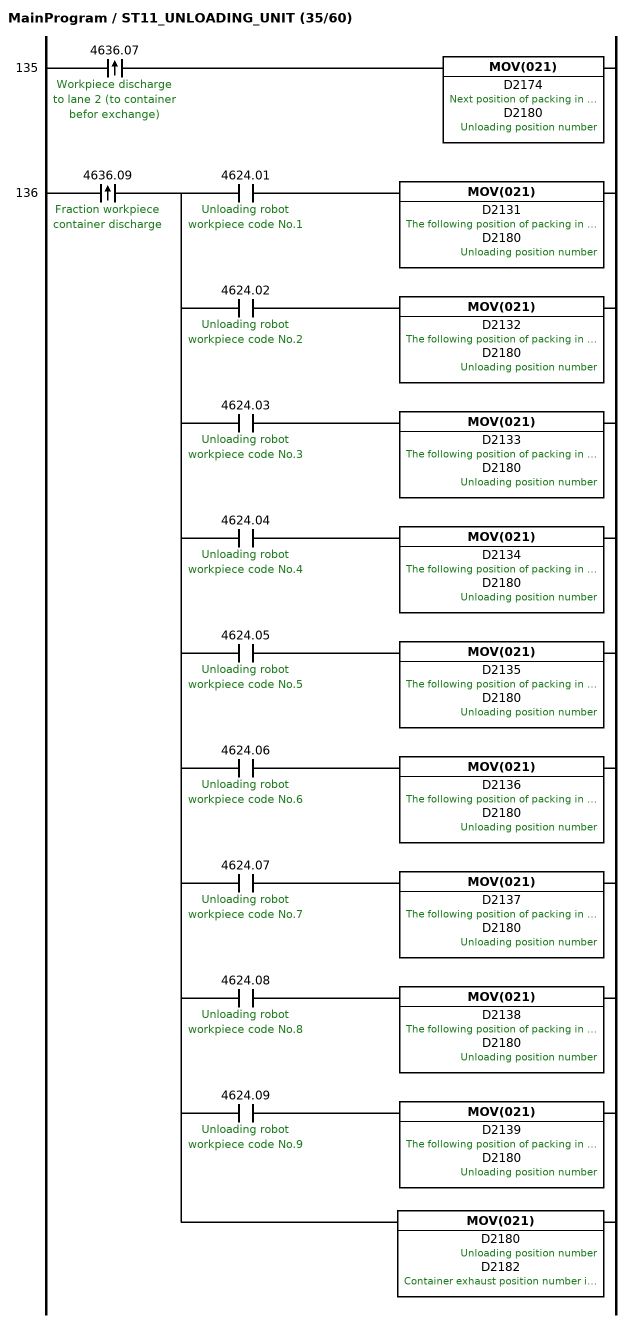
; [picture p552: MainProgram / ST11_UNLOADING_UNIT, rungs 135-136]
; rung 135
@LD 4636.07  ; Workpiece discharge to lane 2 (to container befor exchange)
MOV(021) D2174 D2180  ; Next position of packing in a container of lane 4 (exchange container)(BIN), Unloading position number
; rung 136
@LD 4636.09  ; Fraction workpiece container discharge
OUT TR0
AND 4624.01  ; Unloading robot workpiece code No.1
MOV(021) D2131 D2180  ; The following position of packing in a container number in fraction workpiece (code no.1), Unloading position number
LD TR0
AND 4624.02  ; Unloading robot workpiece code No.2
MOV(021) D2132 D2180  ; The following position of packing in a container number in fraction workpiece (code no.2), Unloading position number
LD TR0
AND 4624.03  ; Unloading robot workpiece code No.3
MOV(021) D2133 D2180  ; The following position of packing in a container number in fraction workpiece (code no.3), Unloading position number
LD TR0
AND 4624.04  ; Unloading robot workpiece code No.4
MOV(021) D2134 D2180  ; The following position of packing in a container number in fraction workpiece (code no.4), Unloading position number
LD TR0
AND 4624.05  ; Unloading robot workpiece code No.5
MOV(021) D2135 D2180  ; The following position of packing in a container number in fraction workpiece (code no.5), Unloading position number
LD TR0
AND 4624.06  ; Unloading robot workpiece code No.6
MOV(021) D2136 D2180  ; The following position of packing in a container number in fraction workpiece (code no.6), Unloading position number
LD TR0
AND 4624.07  ; Unloading robot workpiece code No.7
MOV(021) D2137 D2180  ; The following position of packing in a container number in fraction workpiece (code no.7), Unloading position number
LD TR0
AND 4624.08  ; Unloading robot workpiece code No.8
MOV(021) D2138 D2180  ; The following position of packing in a container number in fraction workpiece (code no.8), Unloading position number
LD TR0
AND 4624.09  ; Unloading robot workpiece code No.9
MOV(021) D2139 D2180  ; The following position of packing in a container number in fraction workpiece (code no.9), Unloading position number
LD TR0
MOV(021) D2180 D2182  ; Unloading position number, Container exhaust position number in fraction workpiece

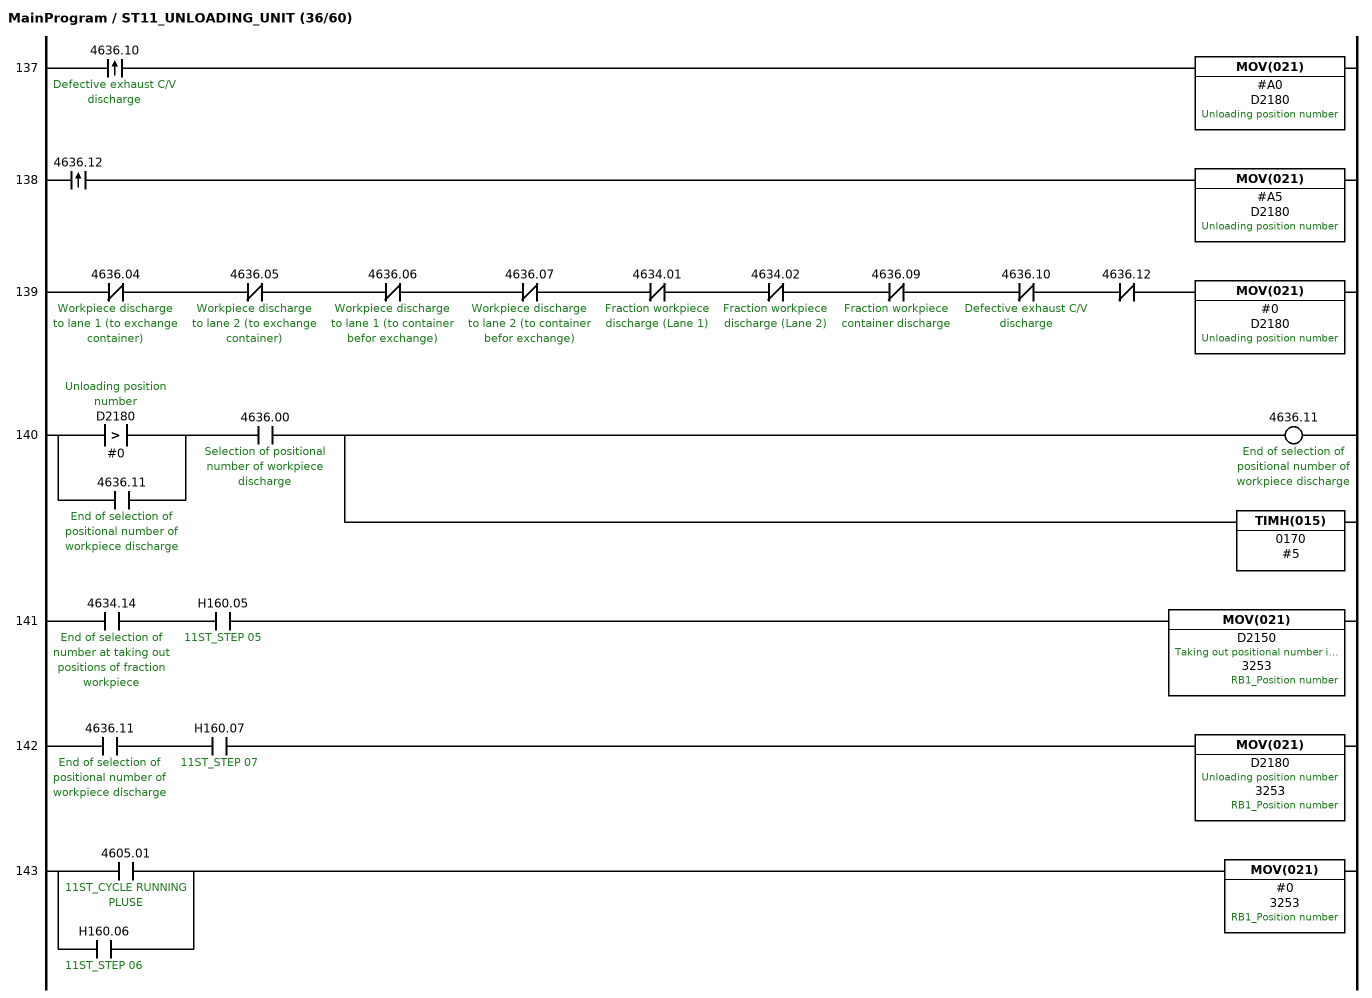
; rung 137
@LD 4636.10  ; Defective exhaust C/V discharge
MOV(021) #A0 D2180  ; Unloading position number
; rung 138
@LD 4636.12
MOV(021) #A5 D2180  ; Unloading position number
; rung 139
LDNOT 4636.04  ; Workpiece discharge to lane 1 (to exchange container)
ANDNOT 4636.05  ; Workpiece discharge to lane 2 (to exchange container)
ANDNOT 4636.06  ; Workpiece discharge to lane 1 (to container befor exchange)
ANDNOT 4636.07  ; Workpiece discharge to lane 2 (to container befor exchange)
ANDNOT 4634.01  ; Fraction workpiece discharge (Lane 1)
ANDNOT 4634.02  ; Fraction workpiece discharge (Lane 2)
ANDNOT 4636.09  ; Fraction workpiece container discharge
ANDNOT 4636.10  ; Defective exhaust C/V discharge
ANDNOT 4636.12
MOV(021) #0 D2180  ; Unloading position number
; rung 140
LD>(320) D2180 #0  ; Unloading position number
OR 4636.11  ; End of selection of positional number of workpiece discharge
AND 4636.00  ; Selection of positional number of workpiece discharge
OUT 4636.11  ; End of selection of positional number of workpiece discharge
TIMH(015) 0170 #5
; rung 141
LD 4634.14  ; End of selection of number at taking out positions of fraction workpiece
AND H160.05  ; 11ST_STEP 05
MOV(021) D2150 3253  ; Taking out positional number in fraction workpiece, RB1_Position number
; rung 142
LD 4636.11  ; End of selection of positional number of workpiece discharge
AND H160.07  ; 11ST_STEP 07
MOV(021) D2180 3253  ; Unloading position number, RB1_Position number
; rung 143
LD 4605.01  ; 11ST_CYCLE RUNNING PLUSE
OR H160.06  ; 11ST_STEP 06
MOV(021) #0 3253  ; RB1_Position number

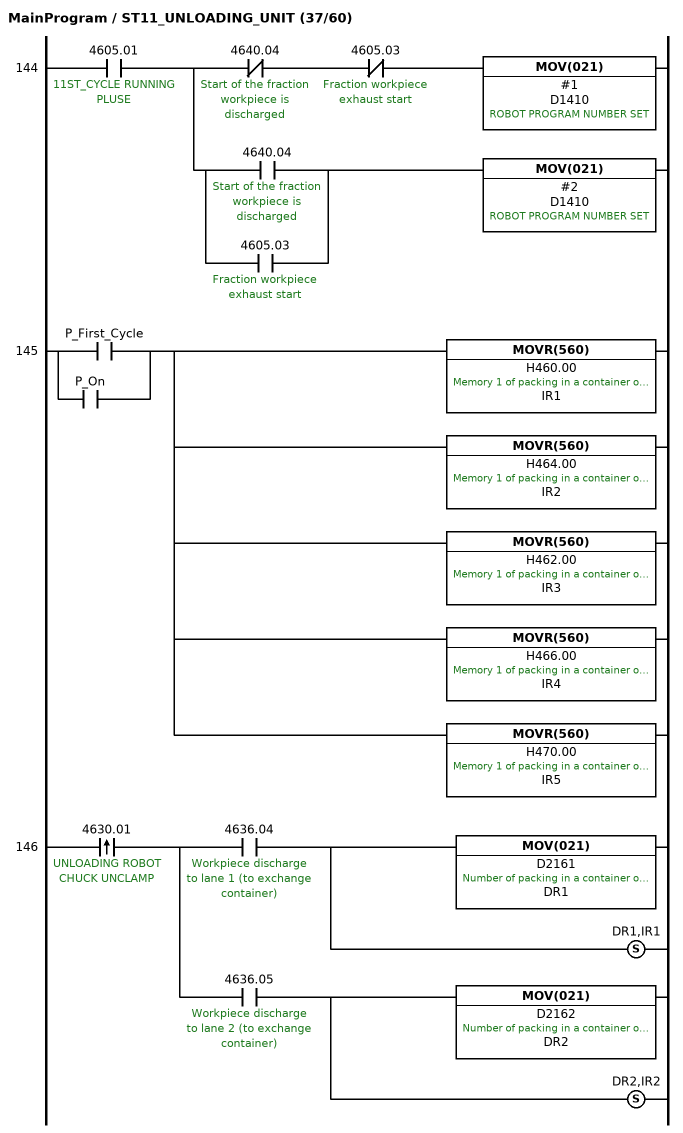
; rung 144
LD 4605.01  ; 11ST_CYCLE RUNNING PLUSE
OUT TR0
ANDNOT 4640.04  ; Start of the fraction workpiece is discharged
ANDNOT 4605.03  ; Fraction workpiece exhaust start
MOV(021) #1 D1410  ; ROBOT PROGRAM NUMBER SET
LD TR0
LD 4640.04  ; Start of the fraction workpiece is discharged
OR 4605.03  ; Fraction workpiece exhaust start
ANDLD
MOV(021) #2 D1410  ; ROBOT PROGRAM NUMBER SET
; rung 145
LD P_First_Cycle
OR P_On  // 様子見で入れた 070619
MOVR(560) H460.00 IR1  ; Memory 1 of packing in a container of lane 1 (exchange container)
MOVR(560) H464.00 IR2  ; Memory 1 of packing in a container of lane 2 (exchange container)
MOVR(560) H462.00 IR3  ; Memory 1 of packing in a container of lane 1 (container befor exchange)
MOVR(560) H466.00 IR4  ; Memory 1 of packing in a container of lane 2 (container befor exchange)
MOVR(560) H470.00 IR5  ; Memory 1 of packing in a container of fraction workpiece
; rung 146
@LD 4630.01  ; UNLOADING ROBOT CHUCK UNCLAMP
OUT TR0
AND 4636.04  ; Workpiece discharge to lane 1 (to exchange container)
MOV(021) D2161 DR1  ; Number of packing in a container of lane 1 (exchange container)(BIN)
SET DR1,IR1
LD TR0
AND 4636.05  ; Workpiece discharge to lane 2 (to exchange container)
MOV(021) D2162 DR2  ; Number of packing in a container of lane 2 (exchange container)(BIN)
SET DR2,IR2

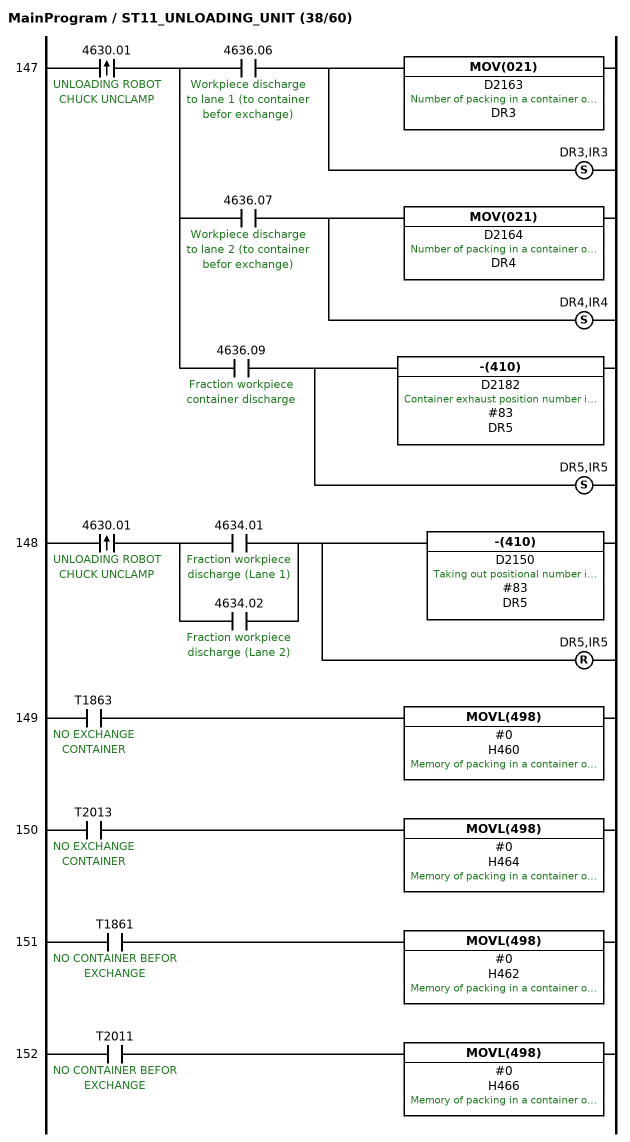
; rung 147
@LD 4630.01  ; UNLOADING ROBOT CHUCK UNCLAMP
OUT TR0
AND 4636.06  ; Workpiece discharge to lane 1 (to container befor exchange)
MOV(021) D2163 DR3  ; Number of packing in a container of lane 1 (container before exchange)(BIN)
SET DR3,IR3
LD TR0
AND 4636.07  ; Workpiece discharge to lane 2 (to container befor exchange)
MOV(021) D2164 DR4  ; Number of packing in a container of lane 2 (container before exchange)(BIN)
SET DR4,IR4
LD TR0
AND 4636.09  ; Fraction workpiece container discharge
-(410) D2182 #83 DR5  ; Container exhaust position number in fraction workpiece
SET DR5,IR5
; rung 148
@LD 4630.01  ; UNLOADING ROBOT CHUCK UNCLAMP
LD 4634.01  ; Fraction workpiece discharge (Lane 1)
OR 4634.02  ; Fraction workpiece discharge (Lane 2)
ANDLD
-(410) D2150 #83 DR5  ; Taking out positional number in fraction workpiece
RSET DR5,IR5
; rung 149
LD T1863  ; NO EXCHANGE CONTAINER
MOVL(498) #0 H460  ; Memory of packing in a container of lane 1 (exchange container)
; rung 150
LD T2013  ; NO EXCHANGE CONTAINER
MOVL(498) #0 H464  ; Memory of packing in a container of lane 2 (exchange container)
; rung 151
LD T1861  ; NO CONTAINER BEFOR EXCHANGE
MOVL(498) #0 H462  ; Memory of packing in a container of lane 1 (container befor exchange)
; rung 152
LD T2011  ; NO CONTAINER BEFOR EXCHANGE
MOVL(498) #0 H466  ; Memory of packing in a container of lane 2 (container befor exchange)

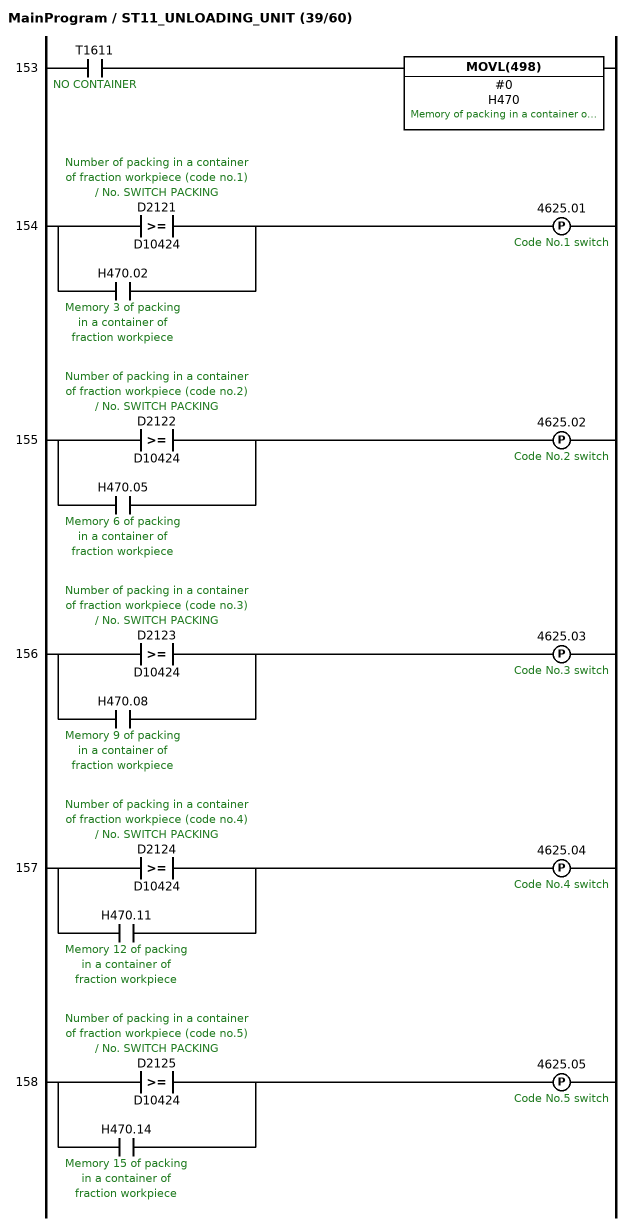
; rung 153
LD T1611  ; NO CONTAINER
MOVL(498) #0 H470  ; Memory of packing in a container of fraction workpiece
; rung 154
LD>=(325) D2121 D10424  ; Number of packing in a container of fraction workpiece (code no.1), No. SWITCH PACKING
OR H470.02  ; Memory 3 of packing in a container of fraction workpiece
DIFU(013) 4625.01  ; Code No.1 switch
; rung 155
LD>=(325) D2122 D10424  ; Number of packing in a container of fraction workpiece (code no.2), No. SWITCH PACKING
OR H470.05  ; Memory 6 of packing in a container of fraction workpiece
DIFU(013) 4625.02  ; Code No.2 switch
; rung 156
LD>=(325) D2123 D10424  ; Number of packing in a container of fraction workpiece (code no.3), No. SWITCH PACKING
OR H470.08  ; Memory 9 of packing in a container of fraction workpiece
DIFU(013) 4625.03  ; Code No.3 switch
; rung 157
LD>=(325) D2124 D10424  ; Number of packing in a container of fraction workpiece (code no.4), No. SWITCH PACKING
OR H470.11  ; Memory 12 of packing in a container of fraction workpiece
DIFU(013) 4625.04  ; Code No.4 switch
; rung 158
LD>=(325) D2125 D10424  ; Number of packing in a container of fraction workpiece (code no.5), No. SWITCH PACKING
OR H470.14  ; Memory 15 of packing in a container of fraction workpiece
DIFU(013) 4625.05  ; Code No.5 switch

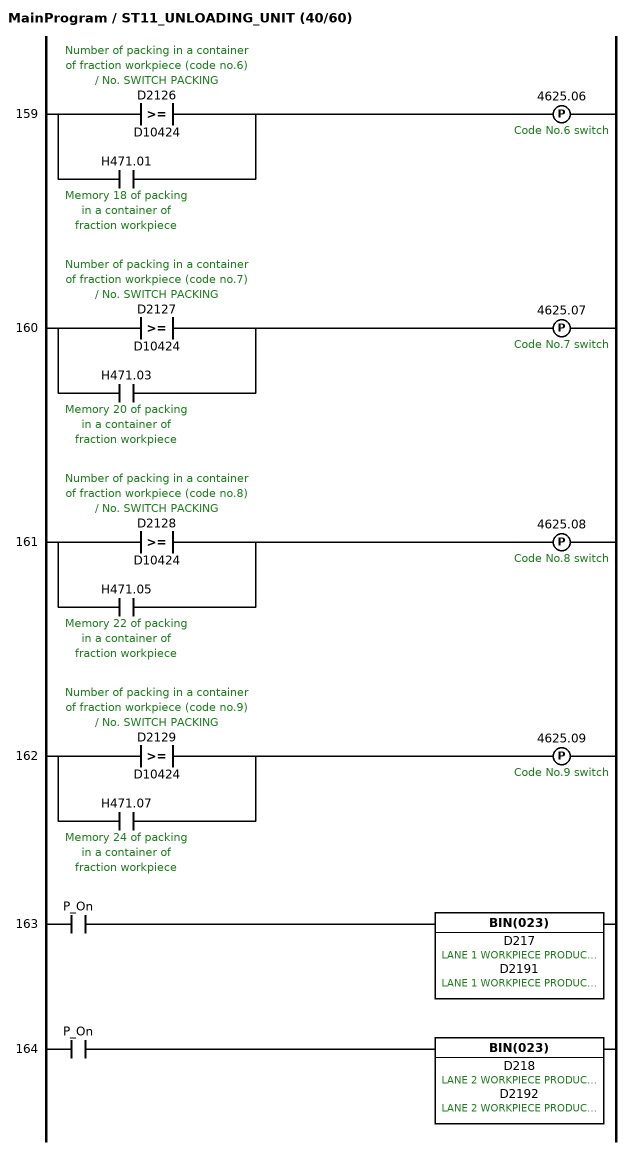
; rung 159
LD>=(325) D2126 D10424  ; Number of packing in a container of fraction workpiece (code no.6), No. SWITCH PACKING
OR H471.01  ; Memory 18 of packing in a container of fraction workpiece
DIFU(013) 4625.06  ; Code No.6 switch
; rung 160
LD>=(325) D2127 D10424  ; Number of packing in a container of fraction workpiece (code no.7), No. SWITCH PACKING
OR H471.03  ; Memory 20 of packing in a container of fraction workpiece
DIFU(013) 4625.07  ; Code No.7 switch
; rung 161
LD>=(325) D2128 D10424  ; Number of packing in a container of fraction workpiece (code no.8), No. SWITCH PACKING
OR H471.05  ; Memory 22 of packing in a container of fraction workpiece
DIFU(013) 4625.08  ; Code No.8 switch
; rung 162
LD>=(325) D2129 D10424  ; Number of packing in a container of fraction workpiece (code no.9), No. SWITCH PACKING
OR H471.07  ; Memory 24 of packing in a container of fraction workpiece
DIFU(013) 4625.09  ; Code No.9 switch
; rung 163
LD P_On
BIN(023) D217 D2191  ; LANE 1 WORKPIECE PRODUCT NUMBER
; rung 164
LD P_On
BIN(023) D218 D2192  ; LANE 2 WORKPIECE PRODUCT NUMBER

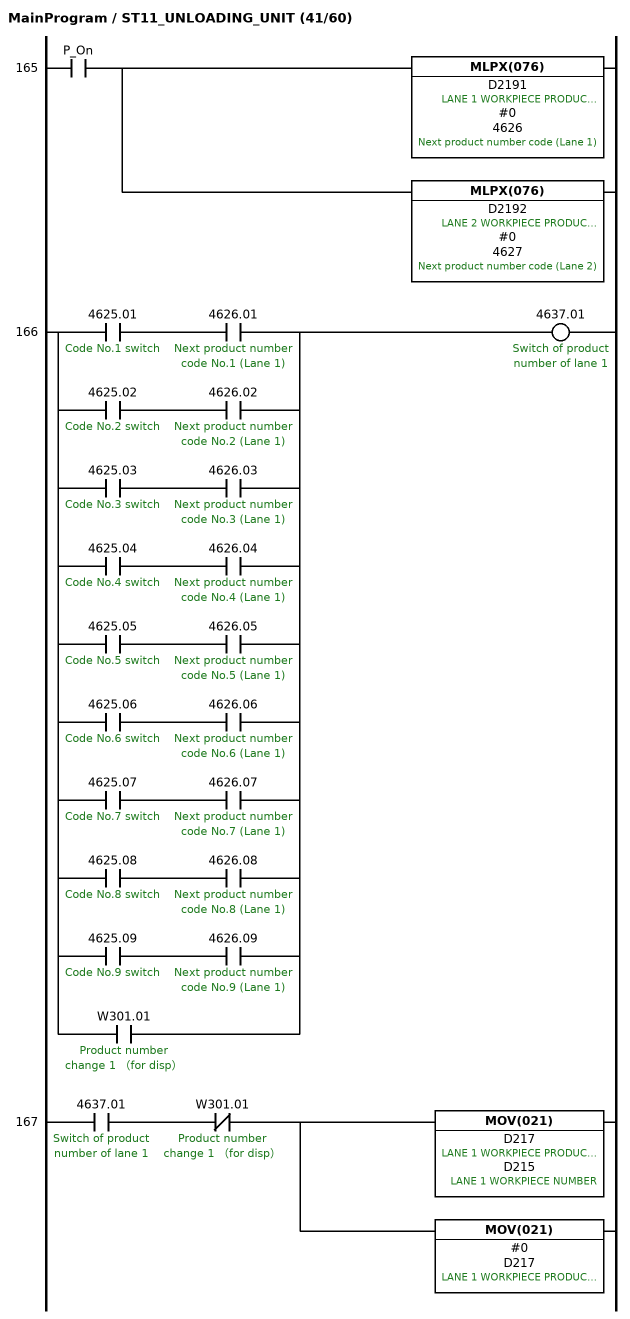
; rung 165
LD P_On
MLPX(076) D2191 #0 4626  ; LANE 1 WORKPIECE PRODUCT NUMBER, Next product number code (Lane 1)
MLPX(076) D2192 #0 4627  ; LANE 2 WORKPIECE PRODUCT NUMBER, Next product number code (Lane 2)
; rung 166
LD 4625.01  ; Code No.1 switch
AND 4626.01  ; Next product number code No.1 (Lane 1)
LD 4625.02  ; Code No.2 switch
AND 4626.02  ; Next product number code No.2 (Lane 1)
ORLD
LD 4625.03  ; Code No.3 switch
AND 4626.03  ; Next product number code No.3 (Lane 1)
ORLD
LD 4625.04  ; Code No.4 switch
AND 4626.04  ; Next product number code No.4 (Lane 1)
ORLD
LD 4625.05  ; Code No.5 switch
AND 4626.05  ; Next product number code No.5 (Lane 1)
ORLD
LD 4625.06  ; Code No.6 switch
AND 4626.06  ; Next product number code No.6 (Lane 1)
ORLD
LD 4625.07  ; Code No.7 switch
AND 4626.07  ; Next product number code No.7 (Lane 1)
ORLD
LD 4625.08  ; Code No.8 switch
AND 4626.08  ; Next product number code No.8 (Lane 1)
ORLD
LD 4625.09  ; Code No.9 switch
AND 4626.09  ; Next product number code No.9 (Lane 1)
ORLD
OR W301.01  ; Product number change 1 （for disp）
OUT 4637.01  ; Switch of product number of lane 1
; rung 167
LD 4637.01  ; Switch of product number of lane 1
ANDNOT W301.01  ; Product number change 1 （for disp）
MOV(021) D217 D215  ; LANE 1 WORKPIECE PRODUCT NUMBER, LANE 1 WORKPIECE NUMBER
MOV(021) #0 D217  ; LANE 1 WORKPIECE PRODUCT NUMBER

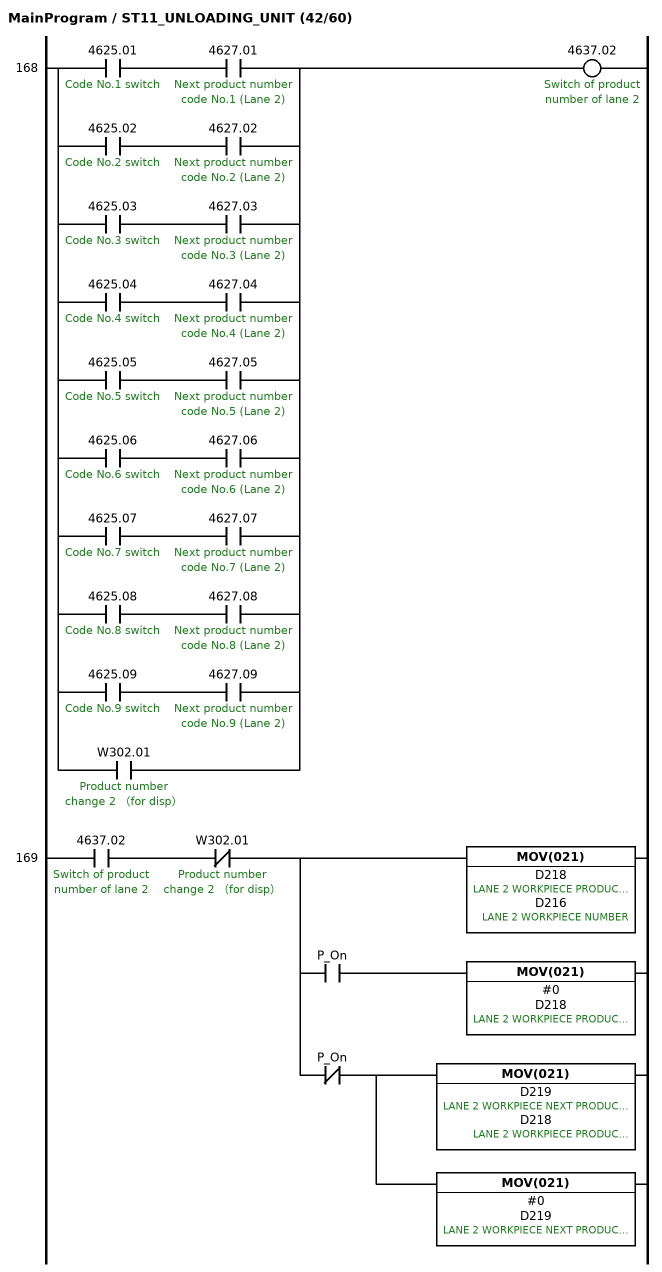
; rung 168
LD 4625.01  ; Code No.1 switch
AND 4627.01  ; Next product number code No.1 (Lane 2)
LD 4625.02  ; Code No.2 switch
AND 4627.02  ; Next product number code No.2 (Lane 2)
ORLD
LD 4625.03  ; Code No.3 switch
AND 4627.03  ; Next product number code No.3 (Lane 2)
ORLD
LD 4625.04  ; Code No.4 switch
AND 4627.04  ; Next product number code No.4 (Lane 2)
ORLD
LD 4625.05  ; Code No.5 switch
AND 4627.05  ; Next product number code No.5 (Lane 2)
ORLD
LD 4625.06  ; Code No.6 switch
AND 4627.06  ; Next product number code No.6 (Lane 2)
ORLD
LD 4625.07  ; Code No.7 switch
AND 4627.07  ; Next product number code No.7 (Lane 2)
ORLD
LD 4625.08  ; Code No.8 switch
AND 4627.08  ; Next product number code No.8 (Lane 2)
ORLD
LD 4625.09  ; Code No.9 switch
AND 4627.09  ; Next product number code No.9 (Lane 2)
ORLD
OR W302.01  ; Product number change 2 （for disp）
OUT 4637.02  ; Switch of product number of lane 2
; rung 169
LD 4637.02  ; Switch of product number of lane 2
ANDNOT W302.01  ; Product number change 2 （for disp）
OUT TR0
MOV(021) D218 D216  ; LANE 2 WORKPIECE PRODUCT NUMBER, LANE 2 WORKPIECE NUMBER
AND P_On
MOV(021) #0 D218  ; LANE 2 WORKPIECE PRODUCT NUMBER
LD TR0
ANDNOT P_On
MOV(021) D219 D218  ; LANE 2 WORKPIECE NEXT PRODUCT NUMBER, LANE 2 WORKPIECE PRODUCT NUMBER
MOV(021) #0 D219  ; LANE 2 WORKPIECE NEXT PRODUCT NUMBER

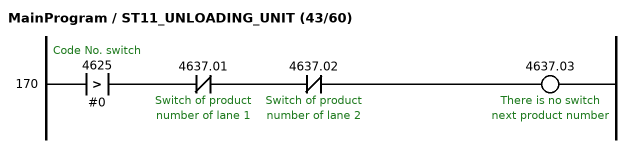
; rung 170
LD>(320) 4625 #0  ; Code No. switch
ANDNOT 4637.01  ; Switch of product number of lane 1
ANDNOT 4637.02  ; Switch of product number of lane 2
OUT 4637.03  ; There is no switch next product number

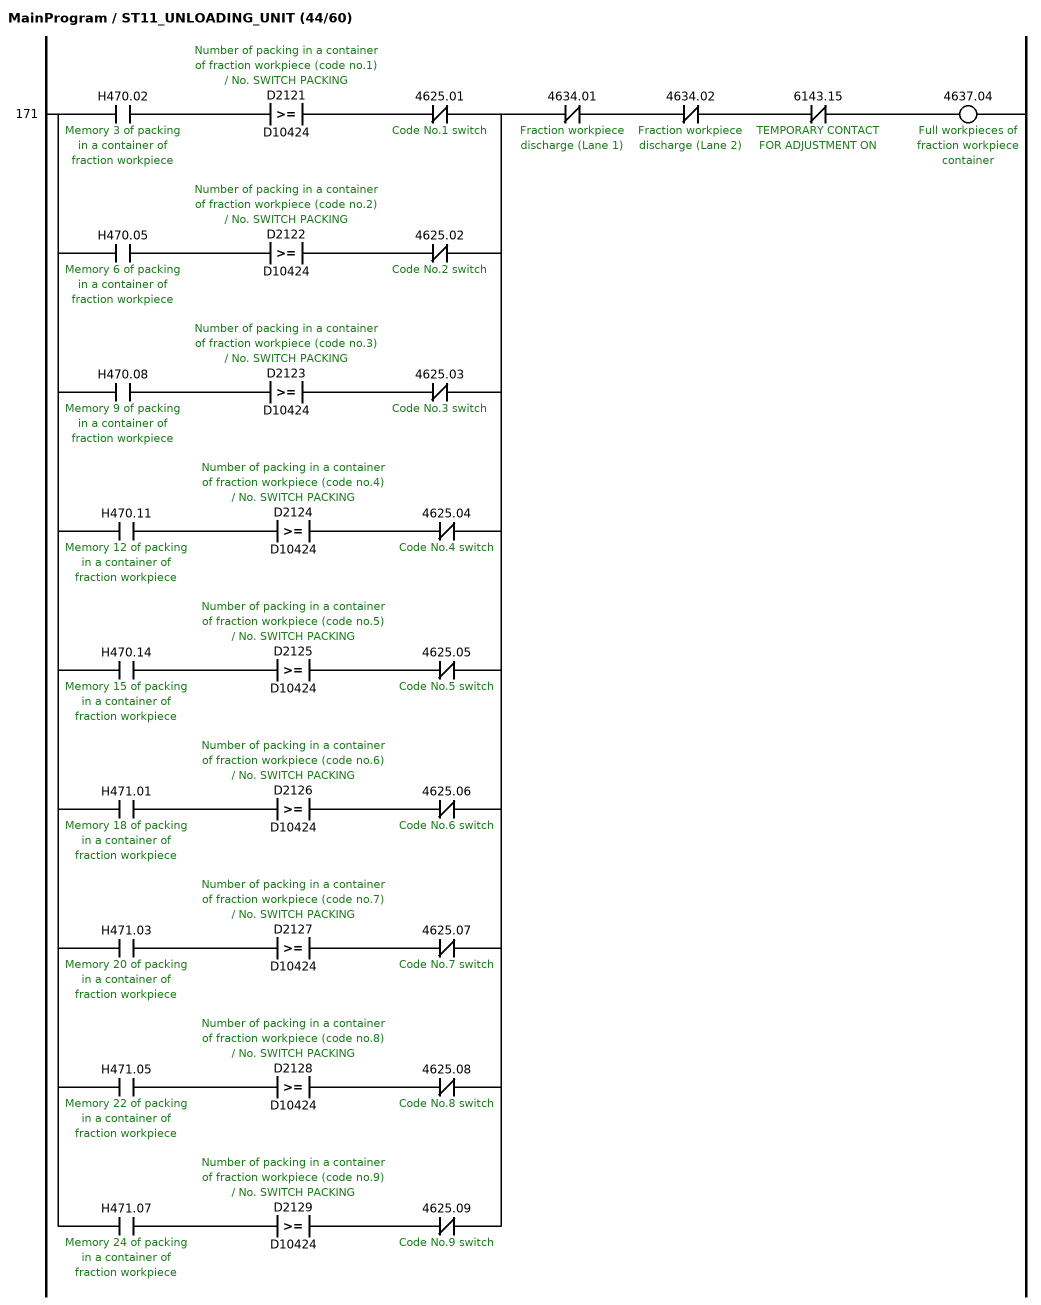
; rung 171
LD H470.02  ; Memory 3 of packing in a container of fraction workpiece
AND>=(325) D2121 D10424  ; Number of packing in a container of fraction workpiece (code no.1), No. SWITCH PACKING
ANDNOT 4625.01  ; Code No.1 switch
LD H470.05  ; Memory 6 of packing in a container of fraction workpiece
AND>=(325) D2122 D10424  ; Number of packing in a container of fraction workpiece (code no.2), No. SWITCH PACKING
ANDNOT 4625.02  ; Code No.2 switch
ORLD
LD H470.08  ; Memory 9 of packing in a container of fraction workpiece
AND>=(325) D2123 D10424  ; Number of packing in a container of fraction workpiece (code no.3), No. SWITCH PACKING
ANDNOT 4625.03  ; Code No.3 switch
ORLD
LD H470.11  ; Memory 12 of packing in a container of fraction workpiece
AND>=(325) D2124 D10424  ; Number of packing in a container of fraction workpiece (code no.4), No. SWITCH PACKING
ANDNOT 4625.04  ; Code No.4 switch
ORLD
LD H470.14  ; Memory 15 of packing in a container of fraction workpiece
AND>=(325) D2125 D10424  ; Number of packing in a container of fraction workpiece (code no.5), No. SWITCH PACKING
ANDNOT 4625.05  ; Code No.5 switch
ORLD
LD H471.01  ; Memory 18 of packing in a container of fraction workpiece
AND>=(325) D2126 D10424  ; Number of packing in a container of fraction workpiece (code no.6), No. SWITCH PACKING
ANDNOT 4625.06  ; Code No.6 switch
ORLD
LD H471.03  ; Memory 20 of packing in a container of fraction workpiece
AND>=(325) D2127 D10424  ; Number of packing in a container of fraction workpiece (code no.7), No. SWITCH PACKING
ANDNOT 4625.07  ; Code No.7 switch
ORLD
LD H471.05  ; Memory 22 of packing in a container of fraction workpiece
AND>=(325) D2128 D10424  ; Number of packing in a container of fraction workpiece (code no.8), No. SWITCH PACKING
ANDNOT 4625.08  ; Code No.8 switch
ORLD
LD H471.07  ; Memory 24 of packing in a container of fraction workpiece
AND>=(325) D2129 D10424  ; Number of packing in a container of fraction workpiece (code no.9), No. SWITCH PACKING
ANDNOT 4625.09  ; Code No.9 switch
ORLD
ANDNOT 4634.01  ; Fraction workpiece discharge (Lane 1)
ANDNOT 4634.02  ; Fraction workpiece discharge (Lane 2)
ANDNOT 6143.15  ; TEMPORARY CONTACT FOR ADJUSTMENT ON
OUT 4637.04  ; Full workpieces of fraction workpiece container

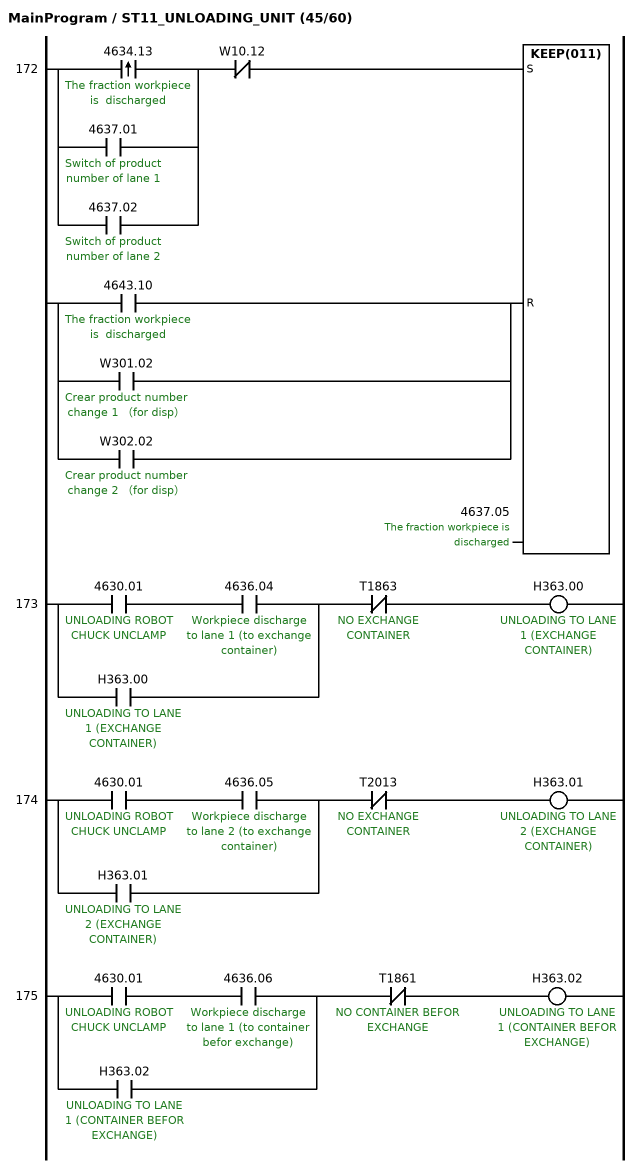
; rung 172
@LD 4634.13  ; The fraction workpiece is  discharged
OR 4637.01  ; Switch of product number of lane 1
OR 4637.02  ; Switch of product number of lane 2
ANDNOT W10.12
LD 4643.10  ; The fraction workpiece is  discharged
OR W301.02  ; Crear product number change 1 （for disp）
OR W302.02  ; Crear product number change 2 （for disp）
KEEP(011) 4637.05  ; The fraction workpiece is  discharged
; rung 173
LD 4630.01  ; UNLOADING ROBOT CHUCK UNCLAMP
AND 4636.04  ; Workpiece discharge to lane 1 (to exchange container)
OR H363.00  ; UNLOADING TO LANE 1 (EXCHANGE CONTAINER)
ANDNOT T1863  ; NO EXCHANGE CONTAINER
OUT H363.00  ; UNLOADING TO LANE 1 (EXCHANGE CONTAINER)
; rung 174
LD 4630.01  ; UNLOADING ROBOT CHUCK UNCLAMP
AND 4636.05  ; Workpiece discharge to lane 2 (to exchange container)
OR H363.01  ; UNLOADING TO LANE 2 (EXCHANGE CONTAINER)
ANDNOT T2013  ; NO EXCHANGE CONTAINER
OUT H363.01  ; UNLOADING TO LANE 2 (EXCHANGE CONTAINER)
; rung 175
LD 4630.01  ; UNLOADING ROBOT CHUCK UNCLAMP
AND 4636.06  ; Workpiece discharge to lane 1 (to container befor exchange)
OR H363.02  ; UNLOADING TO LANE 1 (CONTAINER BEFOR EXCHANGE)
ANDNOT T1861  ; NO CONTAINER BEFOR EXCHANGE
OUT H363.02  ; UNLOADING TO LANE 1 (CONTAINER BEFOR EXCHANGE)

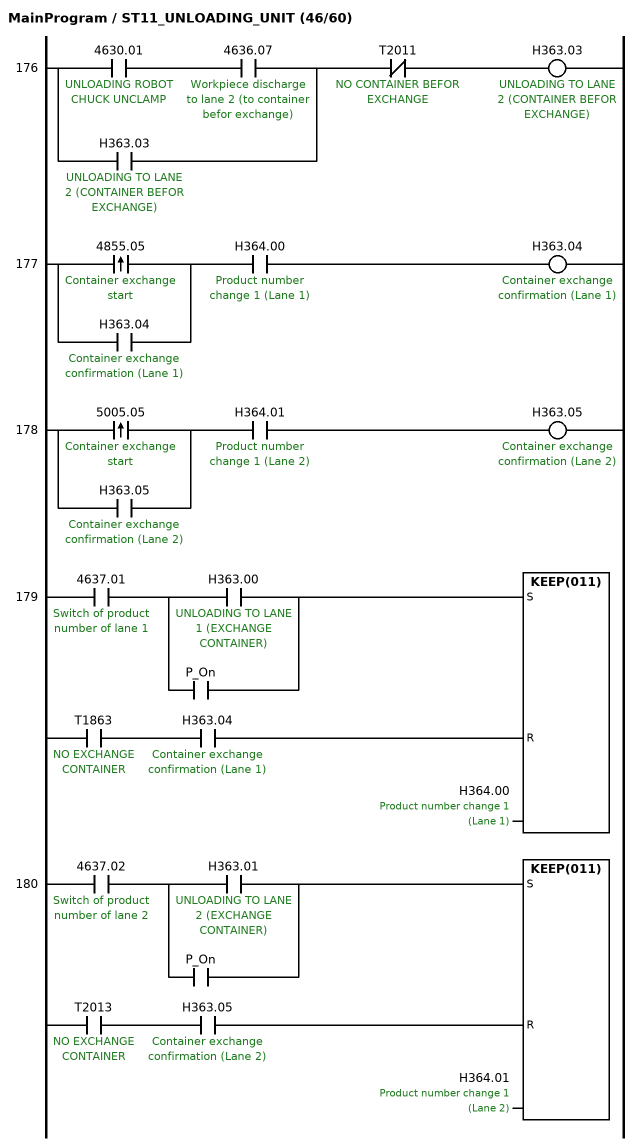
; rung 176
LD 4630.01  ; UNLOADING ROBOT CHUCK UNCLAMP
AND 4636.07  ; Workpiece discharge to lane 2 (to container befor exchange)
OR H363.03  ; UNLOADING TO LANE 2 (CONTAINER BEFOR EXCHANGE)
ANDNOT T2011  ; NO CONTAINER BEFOR EXCHANGE
OUT H363.03  ; UNLOADING TO LANE 2 (CONTAINER BEFOR EXCHANGE)
; rung 177
@LD 4855.05  ; Container exchange start
OR H363.04  ; Container exchange confirmation (Lane 1)
AND H364.00  ; Product number change 1 (Lane 1)
OUT H363.04  ; Container exchange confirmation (Lane 1)
; rung 178
@LD 5005.05  ; Container exchange start
OR H363.05  ; Container exchange confirmation (Lane 2)
AND H364.01  ; Product number change 1 (Lane 2)
OUT H363.05  ; Container exchange confirmation (Lane 2)
; rung 179
LD 4637.01  ; Switch of product number of lane 1
LD H363.00  ; UNLOADING TO LANE 1 (EXCHANGE CONTAINER)
OR P_On
ANDLD
LD T1863  ; NO EXCHANGE CONTAINER
AND H363.04  ; Container exchange confirmation (Lane 1)
KEEP(011) H364.00  ; Product number change 1 (Lane 1)
; rung 180
LD 4637.02  ; Switch of product number of lane 2
LD H363.01  ; UNLOADING TO LANE 2 (EXCHANGE CONTAINER)
OR P_On
ANDLD
LD T2013  ; NO EXCHANGE CONTAINER
AND H363.05  ; Container exchange confirmation (Lane 2)
KEEP(011) H364.01  ; Product number change 1 (Lane 2)

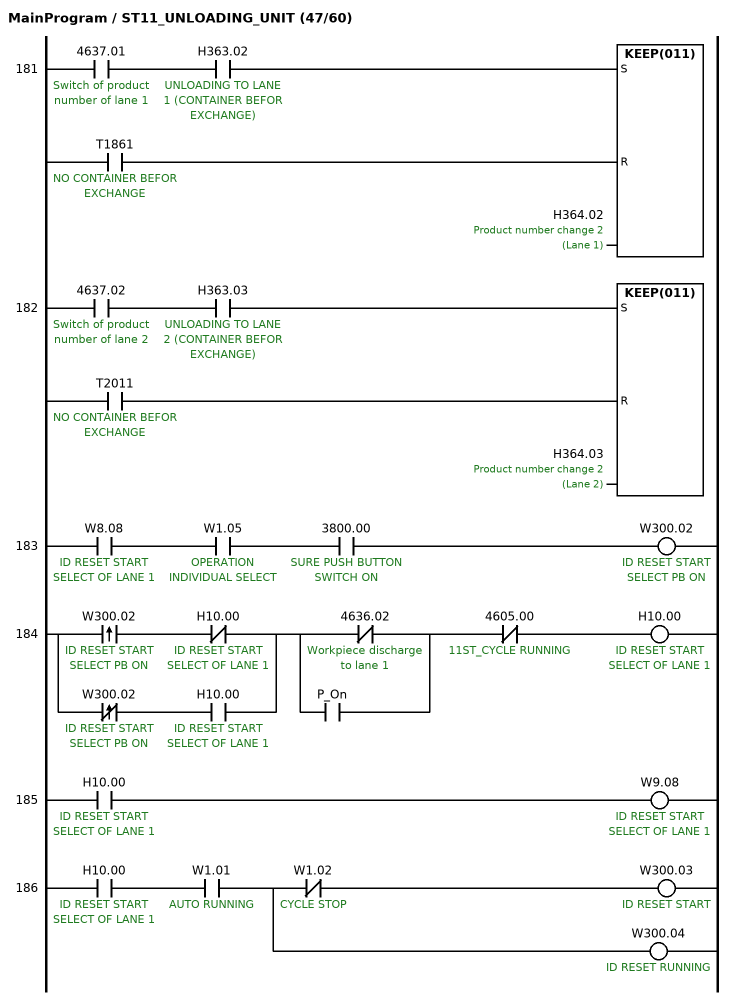
; rung 181
LD 4637.01  ; Switch of product number of lane 1
AND H363.02  ; UNLOADING TO LANE 1 (CONTAINER BEFOR EXCHANGE)
LD T1861  ; NO CONTAINER BEFOR EXCHANGE
KEEP(011) H364.02  ; Product number change 2 (Lane 1)
; rung 182
LD 4637.02  ; Switch of product number of lane 2
AND H363.03  ; UNLOADING TO LANE 2 (CONTAINER BEFOR EXCHANGE)
LD T2011  ; NO CONTAINER BEFOR EXCHANGE
KEEP(011) H364.03  ; Product number change 2 (Lane 2)
; rung 183
LD W8.08  ; ID RESET START SELECT OF LANE 1
AND W1.05  ; OPERATION INDIVIDUAL SELECT
AND 3800.00  ; SURE PUSH BUTTON SWITCH ON
OUT W300.02  ; ID RESET START SELECT PB ON
; rung 184
@LD W300.02  ; ID RESET START SELECT PB ON
ANDNOT H10.00  ; ID RESET START SELECT OF LANE 1
@LDNOT W300.02  ; ID RESET START SELECT PB ON
AND H10.00  ; ID RESET START SELECT OF LANE 1
ORLD
LDNOT 4636.02  ; Workpiece discharge to lane 1
OR P_On
ANDLD
ANDNOT 4605.00  ; 11ST_CYCLE RUNNING
OUT H10.00  ; ID RESET START SELECT OF LANE 1
; rung 185
LD H10.00  ; ID RESET START SELECT OF LANE 1
OUT W9.08  ; ID RESET START SELECT OF LANE 1
; rung 186
LD H10.00  ; ID RESET START SELECT OF LANE 1
AND W1.01  ; AUTO RUNNING
OUT TR0
ANDNOT W1.02  ; CYCLE STOP
OUT W300.03  ; ID RESET START
LD TR0
OUT W300.04  ; ID RESET RUNNING

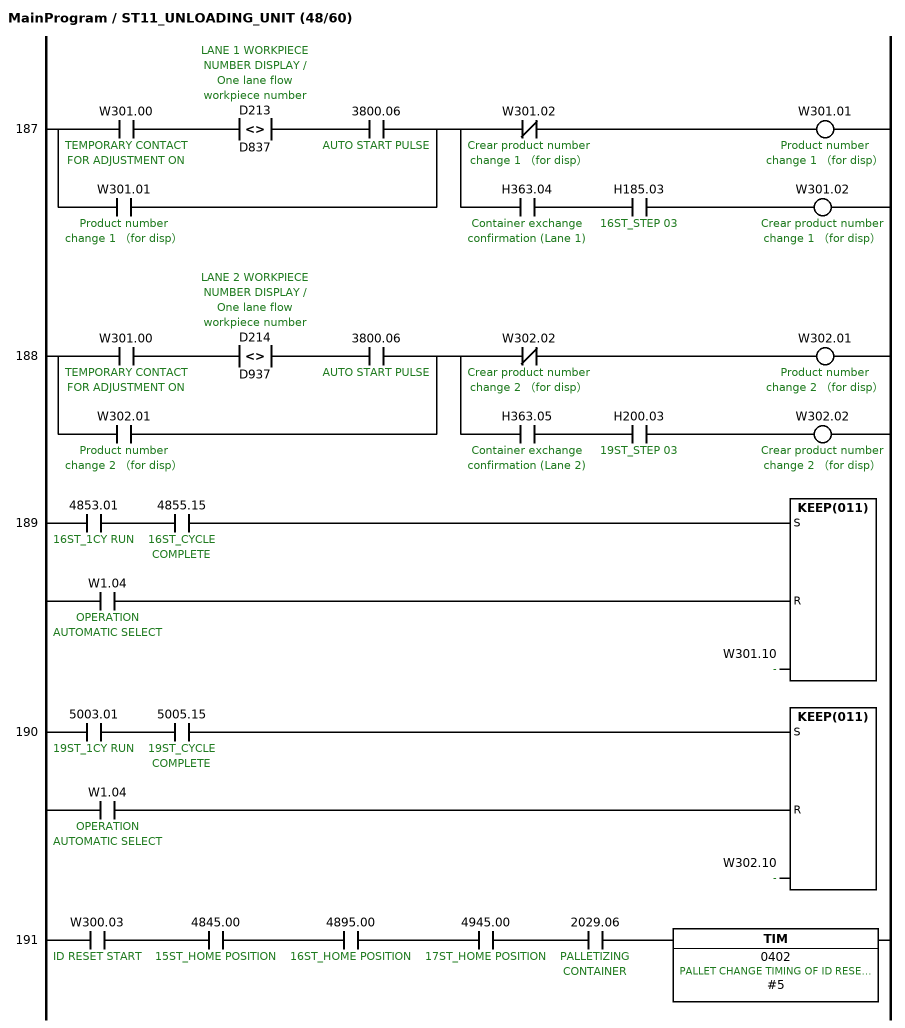
; rung 187
LD W301.00  ; TEMPORARY CONTACT FOR ADJUSTMENT ON
AND<>(305) D213 D837  ; LANE 1 WORKPIECE NUMBER DISPLAY, One lane flow workpiece number
AND 3800.06  ; AUTO START PULSE
OR W301.01  ; Product number change 1 （for disp）
OUT TR0
ANDNOT W301.02  ; Crear product number change 1 （for disp）
OUT W301.01  ; Product number change 1 （for disp）
LD TR0
AND H363.04  ; Container exchange confirmation (Lane 1)
AND H185.03  ; 16ST_STEP 03
OUT W301.02  ; Crear product number change 1 （for disp）
; rung 188
LD W301.00  ; TEMPORARY CONTACT FOR ADJUSTMENT ON
AND<>(305) D214 D937  ; LANE 2 WORKPIECE NUMBER DISPLAY, One lane flow workpiece number
AND 3800.06  ; AUTO START PULSE
OR W302.01  ; Product number change 2 （for disp）
OUT TR0
ANDNOT W302.02  ; Crear product number change 2 （for disp）
OUT W302.01  ; Product number change 2 （for disp）
LD TR0
AND H363.05  ; Container exchange confirmation (Lane 2)
AND H200.03  ; 19ST_STEP 03
OUT W302.02  ; Crear product number change 2 （for disp）
; rung 189
LD 4853.01  ; 16ST_1CY RUN
AND 4855.15  ; 16ST_CYCLE COMPLETE
LD W1.04  ; OPERATION AUTOMATIC SELECT
KEEP(011) W301.10  ; -
; rung 190
LD 5003.01  ; 19ST_1CY RUN
AND 5005.15  ; 19ST_CYCLE COMPLETE
LD W1.04  ; OPERATION AUTOMATIC SELECT
KEEP(011) W302.10  ; -
; rung 191
LD W300.03  ; ID RESET START
AND 4845.00  ; 15ST_HOME POSITION
AND 4895.00  ; 16ST_HOME POSITION
AND 4945.00  ; 17ST_HOME POSITION
AND 2029.06  ; PALLETIZING CONTAINER
TIM 0402 #5  ; PALLET CHANGE TIMING OF ID RESET START SELECT

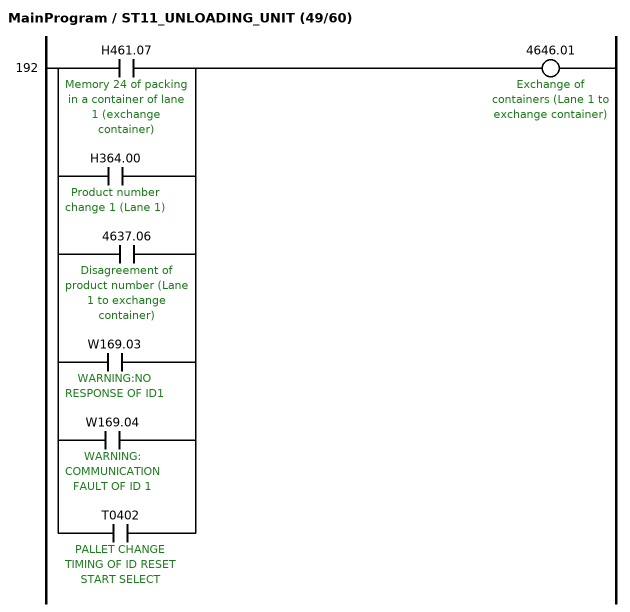
; rung 192
LD H461.07  ; Memory 24 of packing in a container of lane 1 (exchange container)
OR H364.00  ; Product number change 1 (Lane 1)
OR 4637.06  ; Disagreement of product number (Lane 1 to exchange container)
OR W169.03  ; WARNING:NO RESPONSE OF ID1
OR W169.04  ; WARNING:COMMUNICATION FAULT OF ID 1
OR T0402  ; PALLET CHANGE TIMING OF ID RESET START SELECT
OUT 4646.01  ; Exchange of containers (Lane 1 to exchange container)

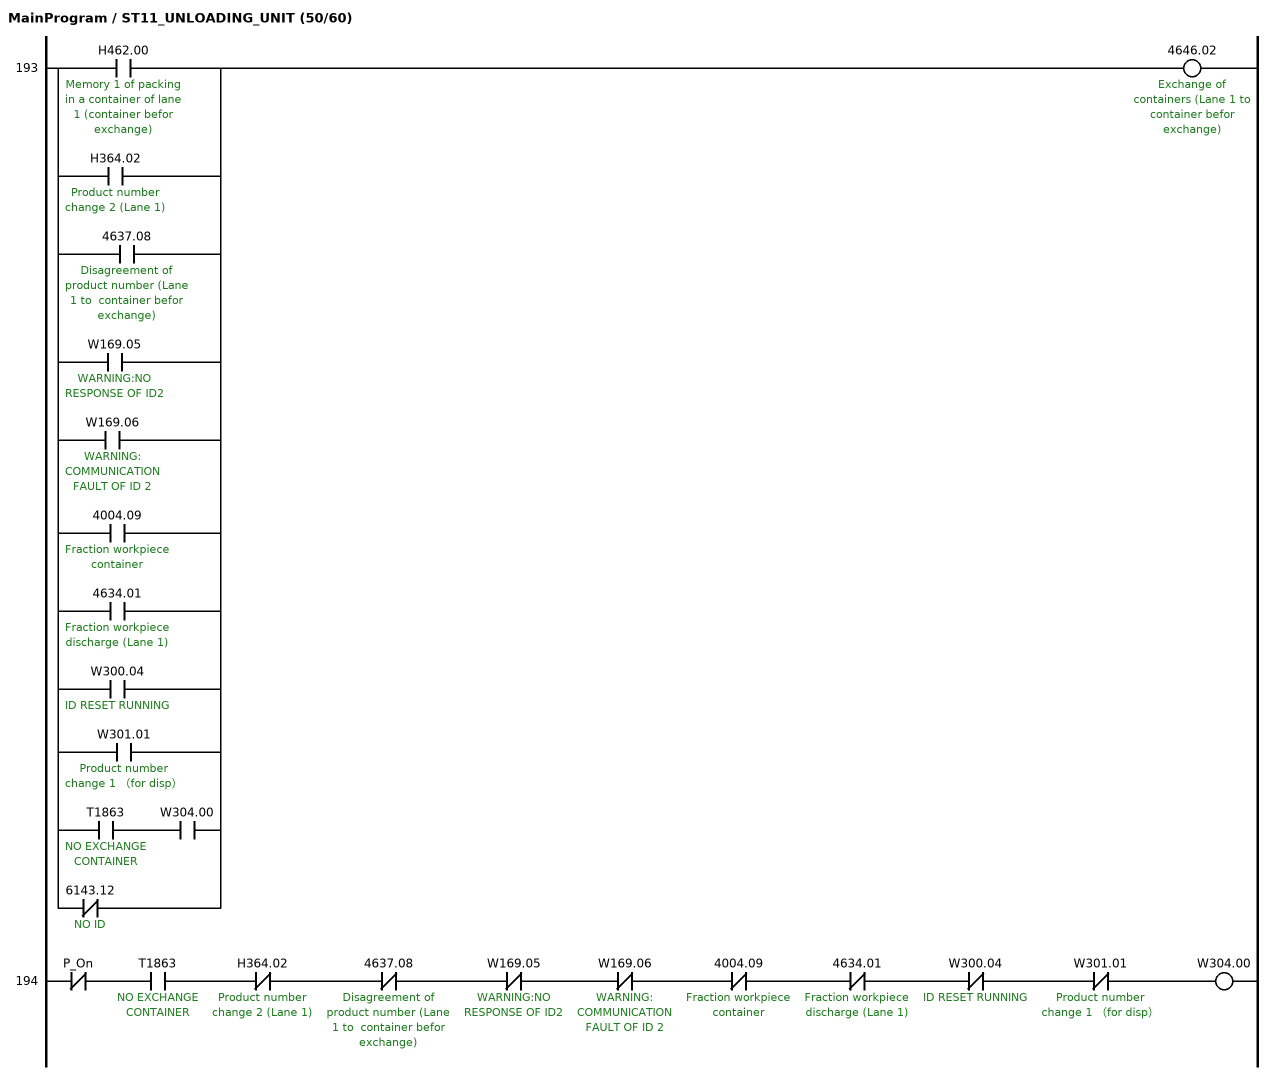
; rung 193
LD H462.00  ; Memory 1 of packing in a container of lane 1 (container befor exchange)
OR H364.02  ; Product number change 2 (Lane 1)
OR 4637.08  ; Disagreement of product number (Lane 1 to  container befor exchange)
OR W169.05  ; WARNING:NO RESPONSE OF ID2
OR W169.06  ; WARNING:COMMUNICATION FAULT OF ID 2
OR 4004.09  ; Fraction workpiece container
OR 4634.01  ; Fraction workpiece discharge (Lane 1)
OR W300.04  ; ID RESET RUNNING
OR W301.01  ; Product number change 1 （for disp）
LD T1863  ; NO EXCHANGE CONTAINER
AND W304.00
ORLD
ORNOT 6143.12  ; NO ID
OUT 4646.02  ; Exchange of containers (Lane 1 to container befor exchange)
; rung 194
LDNOT P_On
AND T1863  ; NO EXCHANGE CONTAINER
ANDNOT H364.02  ; Product number change 2 (Lane 1)
ANDNOT 4637.08  ; Disagreement of product number (Lane 1 to  container befor exchange)
ANDNOT W169.05  ; WARNING:NO RESPONSE OF ID2
ANDNOT W169.06  ; WARNING:COMMUNICATION FAULT OF ID 2
ANDNOT 4004.09  ; Fraction workpiece container
ANDNOT 4634.01  ; Fraction workpiece discharge (Lane 1)
ANDNOT W300.04  ; ID RESET RUNNING
ANDNOT W301.01  ; Product number change 1 （for disp）
OUT W304.00

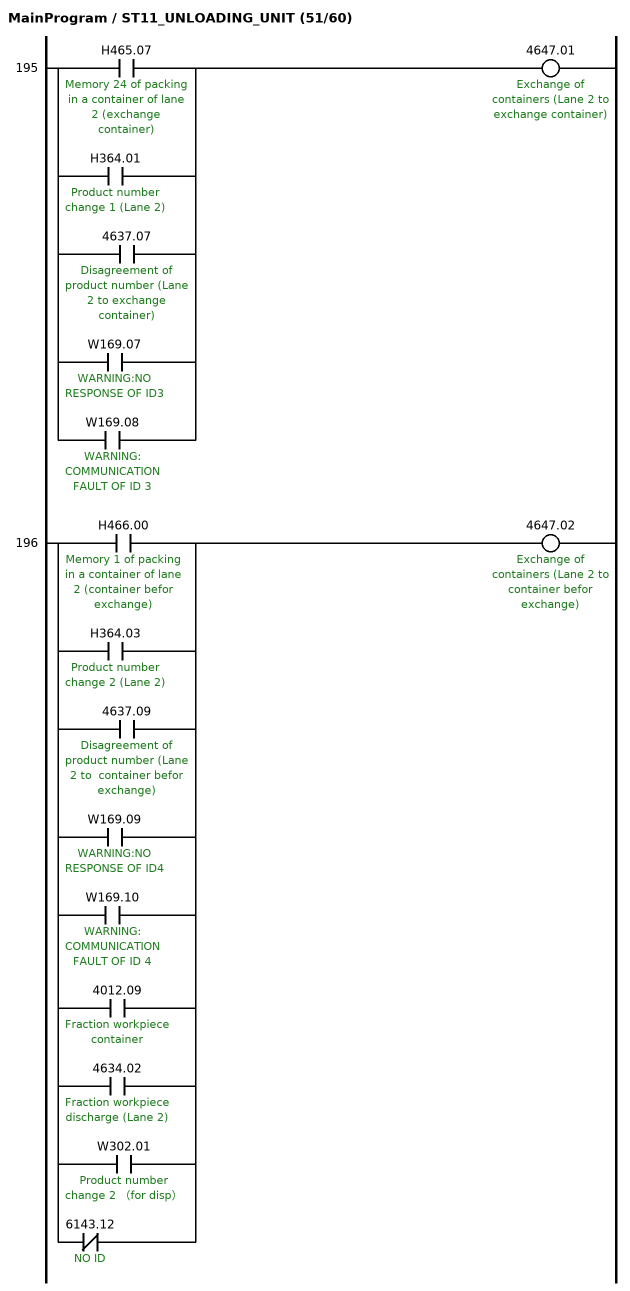
; rung 195
LD H465.07  ; Memory 24 of packing in a container of lane 2 (exchange container)
OR H364.01  ; Product number change 1 (Lane 2)
OR 4637.07  ; Disagreement of product number (Lane 2 to exchange container)
OR W169.07  ; WARNING:NO RESPONSE OF ID3
OR W169.08  ; WARNING:COMMUNICATION FAULT OF ID 3
OUT 4647.01  ; Exchange of containers (Lane 2 to exchange container)
; rung 196
LD H466.00  ; Memory 1 of packing in a container of lane 2 (container befor exchange)
OR H364.03  ; Product number change 2 (Lane 2)
OR 4637.09  ; Disagreement of product number (Lane 2 to  container befor exchange)
OR W169.09  ; WARNING:NO RESPONSE OF ID4
OR W169.10  ; WARNING:COMMUNICATION FAULT OF ID 4
OR 4012.09  ; Fraction workpiece container
OR 4634.02  ; Fraction workpiece discharge (Lane 2)
OR W302.01  ; Product number change 2 （for disp）
ORNOT 6143.12  ; NO ID
OUT 4647.02  ; Exchange of containers (Lane 2 to container befor exchange)

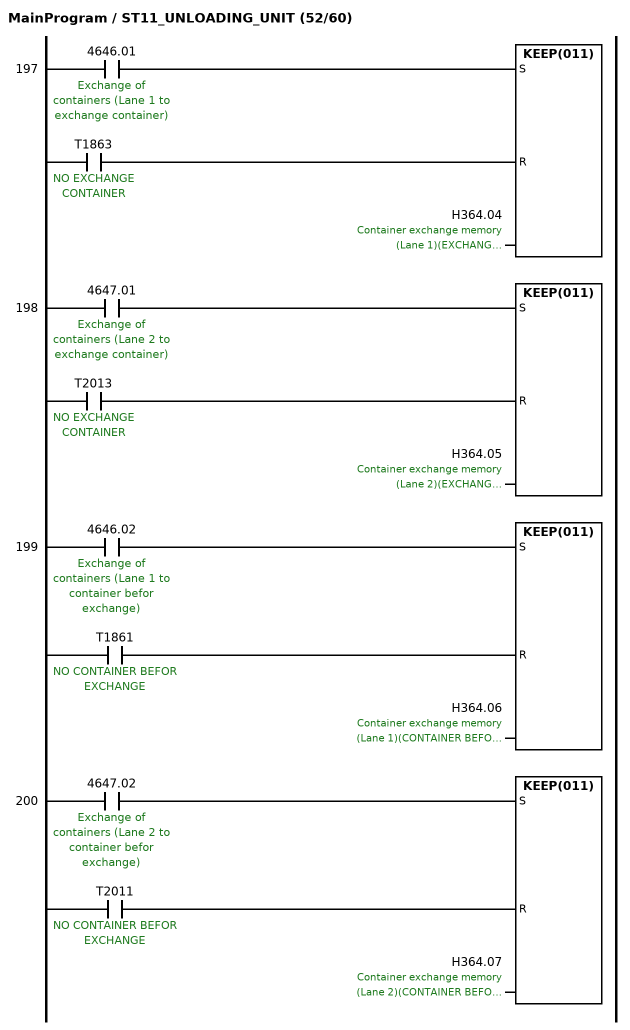
; rung 197
LD 4646.01  ; Exchange of containers (Lane 1 to exchange container)
LD T1863  ; NO EXCHANGE CONTAINER
KEEP(011) H364.04  ; Container exchange memory (Lane 1)(EXCHANGE CONTAINER)
; rung 198
LD 4647.01  ; Exchange of containers (Lane 2 to exchange container)
LD T2013  ; NO EXCHANGE CONTAINER
KEEP(011) H364.05  ; Container exchange memory (Lane 2)(EXCHANGE CONTAINER)
; rung 199
LD 4646.02  ; Exchange of containers (Lane 1 to container befor exchange)
LD T1861  ; NO CONTAINER BEFOR EXCHANGE
KEEP(011) H364.06  ; Container exchange memory (Lane 1)(CONTAINER BEFOR EXCHANGE)
; rung 200
LD 4647.02  ; Exchange of containers (Lane 2 to container befor exchange)
LD T2011  ; NO CONTAINER BEFOR EXCHANGE
KEEP(011) H364.07  ; Container exchange memory (Lane 2)(CONTAINER BEFOR EXCHANGE)

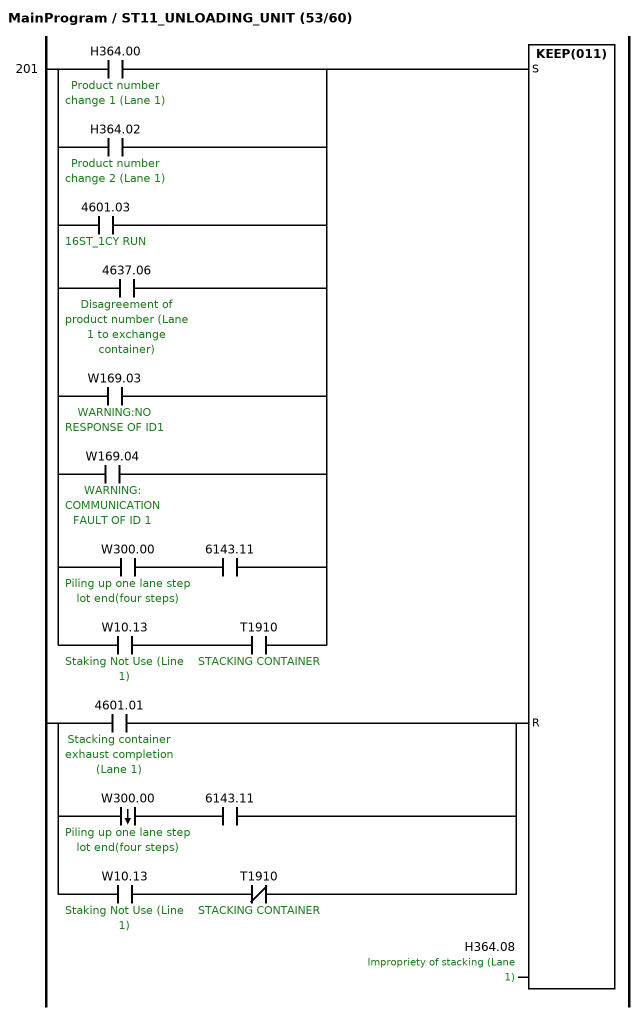
; rung 201
LD H364.00  ; Product number change 1 (Lane 1)
OR H364.02  ; Product number change 2 (Lane 1)
OR 4601.03  ; 16ST_1CY RUN
OR 4637.06  ; Disagreement of product number (Lane 1 to exchange container)
OR W169.03  ; WARNING:NO RESPONSE OF ID1
OR W169.04  ; WARNING:COMMUNICATION FAULT OF ID 1
LD W300.00  ; Piling up one lane step lot end(four steps)
AND 6143.11
ORLD
LD W10.13  ; Staking Not Use (Line 1)
AND T1910  ; STACKING CONTAINER
ORLD
LD 4601.01  ; Stacking container exhaust completion (Lane 1)
%LD W300.00  ; Piling up one lane step lot end(four steps)
AND 6143.11
ORLD
LD W10.13  ; Staking Not Use (Line 1)
ANDNOT T1910  ; STACKING CONTAINER
ORLD
KEEP(011) H364.08  ; Impropriety of stacking (Lane 1)

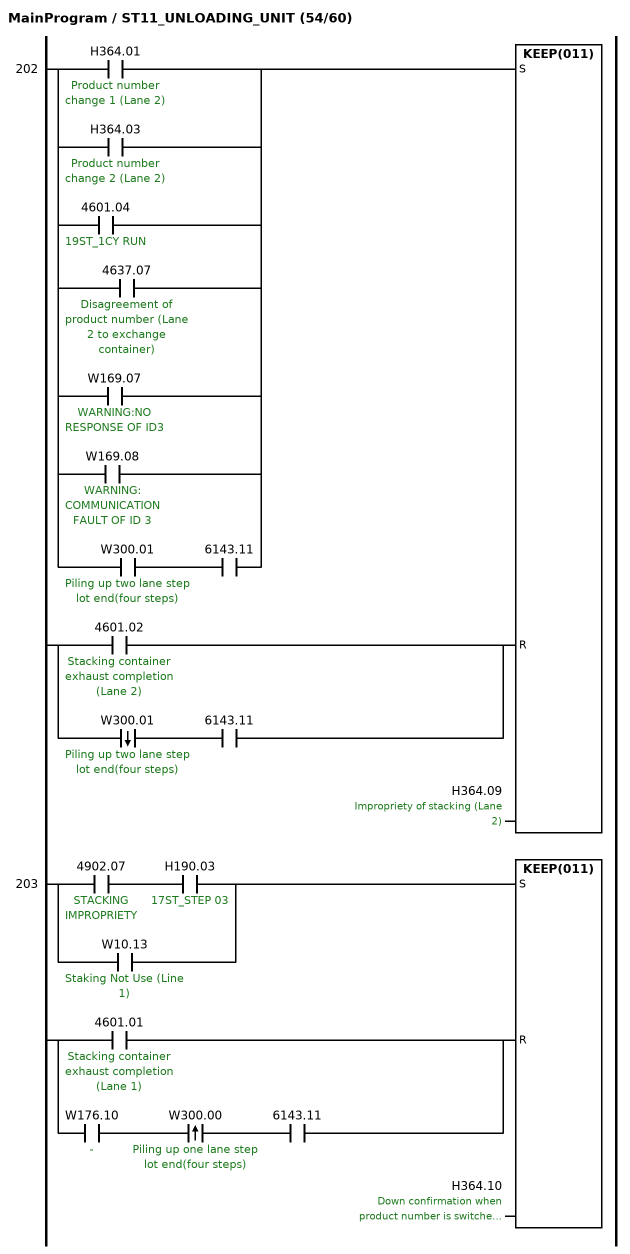
; rung 202
LD H364.01  ; Product number change 1 (Lane 2)
OR H364.03  ; Product number change 2 (Lane 2)
OR 4601.04  ; 19ST_1CY RUN
OR 4637.07  ; Disagreement of product number (Lane 2 to exchange container)
OR W169.07  ; WARNING:NO RESPONSE OF ID3
OR W169.08  ; WARNING:COMMUNICATION FAULT OF ID 3
LD W300.01  ; Piling up two lane step lot end(four steps)
AND 6143.11
ORLD
LD 4601.02  ; Stacking container exhaust completion (Lane 2)
%LD W300.01  ; Piling up two lane step lot end(four steps)
AND 6143.11
ORLD
KEEP(011) H364.09  ; Impropriety of stacking (Lane 2)
; rung 203
LD 4902.07  ; STACKING IMPROPRIETY
AND H190.03  ; 17ST_STEP 03
OR W10.13  ; Staking Not Use (Line 1)
LD 4601.01  ; Stacking container exhaust completion (Lane 1)
LD W176.10  ; -
@AND W300.00  ; Piling up one lane step lot end(four steps)
AND 6143.11
ORLD
KEEP(011) H364.10  ; Down confirmation when product number is switched (Lane 1)

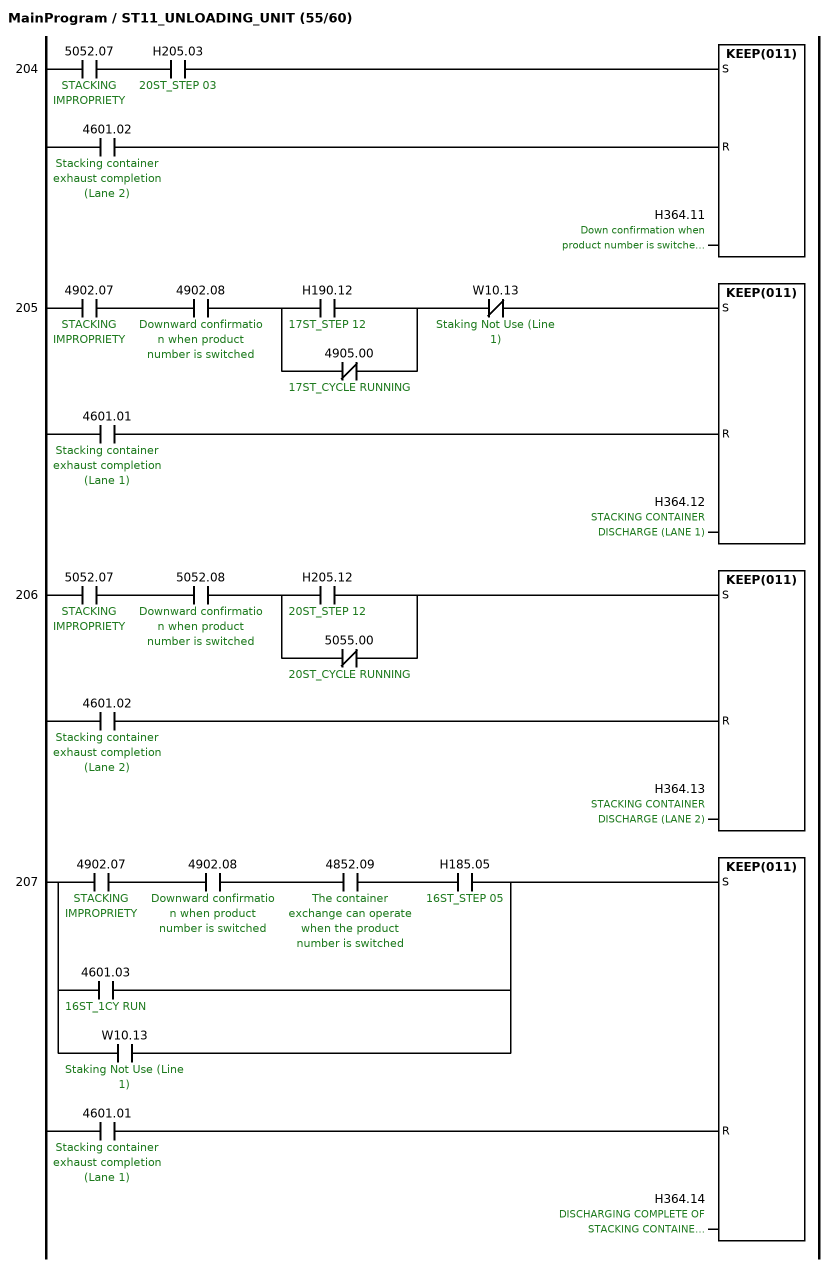
; rung 204
LD 5052.07  ; STACKING IMPROPRIETY
AND H205.03  ; 20ST_STEP 03
LD 4601.02  ; Stacking container exhaust completion (Lane 2)
KEEP(011) H364.11  ; Down confirmation when product number is switched (Lane 2)
; rung 205
LD 4902.07  ; STACKING IMPROPRIETY
AND 4902.08  ; Downward confirmation when product number is switched
LD H190.12  ; 17ST_STEP 12
ORNOT 4905.00  ; 17ST_CYCLE RUNNING
ANDLD
ANDNOT W10.13  ; Staking Not Use (Line 1)
LD 4601.01  ; Stacking container exhaust completion (Lane 1)
KEEP(011) H364.12  ; STACKING CONTAINER DISCHARGE (LANE 1)
; rung 206
LD 5052.07  ; STACKING IMPROPRIETY
AND 5052.08  ; Downward confirmation when product number is switched
LD H205.12  ; 20ST_STEP 12
ORNOT 5055.00  ; 20ST_CYCLE RUNNING
ANDLD
LD 4601.02  ; Stacking container exhaust completion (Lane 2)
KEEP(011) H364.13  ; STACKING CONTAINER DISCHARGE (LANE 2)
; rung 207
LD 4902.07  ; STACKING IMPROPRIETY
AND 4902.08  ; Downward confirmation when product number is switched
AND 4852.09  ; The container exchange can operate when the product number is switched
AND H185.05  ; 16ST_STEP 05
OR 4601.03  ; 16ST_1CY RUN
OR W10.13  ; Staking Not Use (Line 1)
LD 4601.01  ; Stacking container exhaust completion (Lane 1)
KEEP(011) H364.14  ; DISCHARGING COMPLETE OF STACKING CONTAINER  (LANE 1)

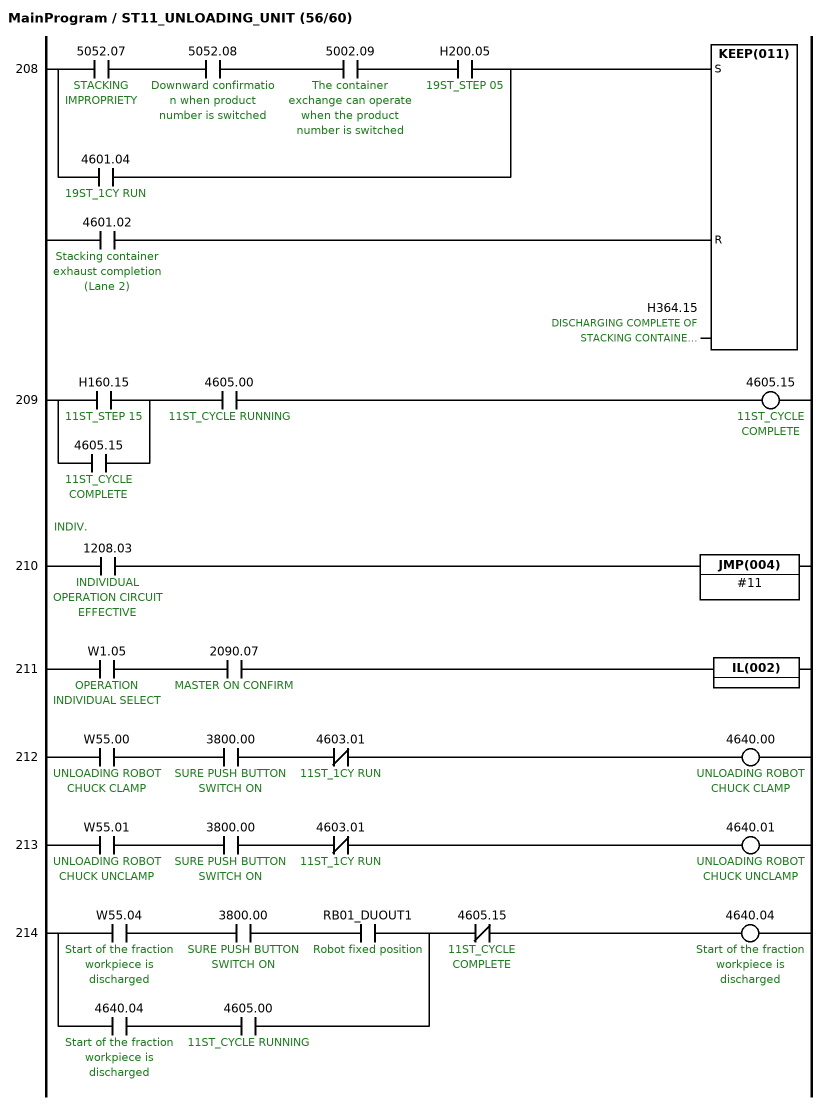
; rung 208
LD 5052.07  ; STACKING IMPROPRIETY
AND 5052.08  ; Downward confirmation when product number is switched
AND 5002.09  ; The container exchange can operate when the product number is switched
AND H200.05  ; 19ST_STEP 05
OR 4601.04  ; 19ST_1CY RUN
LD 4601.02  ; Stacking container exhaust completion (Lane 2)
KEEP(011) H364.15  ; DISCHARGING COMPLETE OF STACKING CONTAINER  (LANE 2)
; rung 209
LD H160.15  ; 11ST_STEP 15
OR 4605.15  ; 11ST_CYCLE COMPLETE
AND 4605.00  ; 11ST_CYCLE RUNNING
OUT 4605.15  ; 11ST_CYCLE COMPLETE
; rung 210: INDIV.
LD 1208.03  ; INDIVIDUAL OPERATION CIRCUIT EFFECTIVE
JMP(004) #11
; rung 211
LD W1.05  ; OPERATION INDIVIDUAL SELECT
AND 2090.07  ; MASTER ON CONFIRM
IL(002)
; rung 212
LD W55.00  ; UNLOADING ROBOT CHUCK CLAMP
AND 3800.00  ; SURE PUSH BUTTON SWITCH ON
ANDNOT 4603.01  ; 11ST_1CY RUN
OUT 4640.00  ; UNLOADING ROBOT CHUCK CLAMP
; rung 213
LD W55.01  ; UNLOADING ROBOT CHUCK UNCLAMP
AND 3800.00  ; SURE PUSH BUTTON SWITCH ON
ANDNOT 4603.01  ; 11ST_1CY RUN
OUT 4640.01  ; UNLOADING ROBOT CHUCK UNCLAMP
; rung 214
LD W55.04  ; Start of the fraction workpiece is discharged
AND 3800.00  ; SURE PUSH BUTTON SWITCH ON
AND RB01_DUOUT1  ; Robot fixed position
LD 4640.04  ; Start of the fraction workpiece is discharged
AND 4605.00  ; 11ST_CYCLE RUNNING
ORLD
ANDNOT 4605.15  ; 11ST_CYCLE COMPLETE
OUT 4640.04  ; Start of the fraction workpiece is discharged

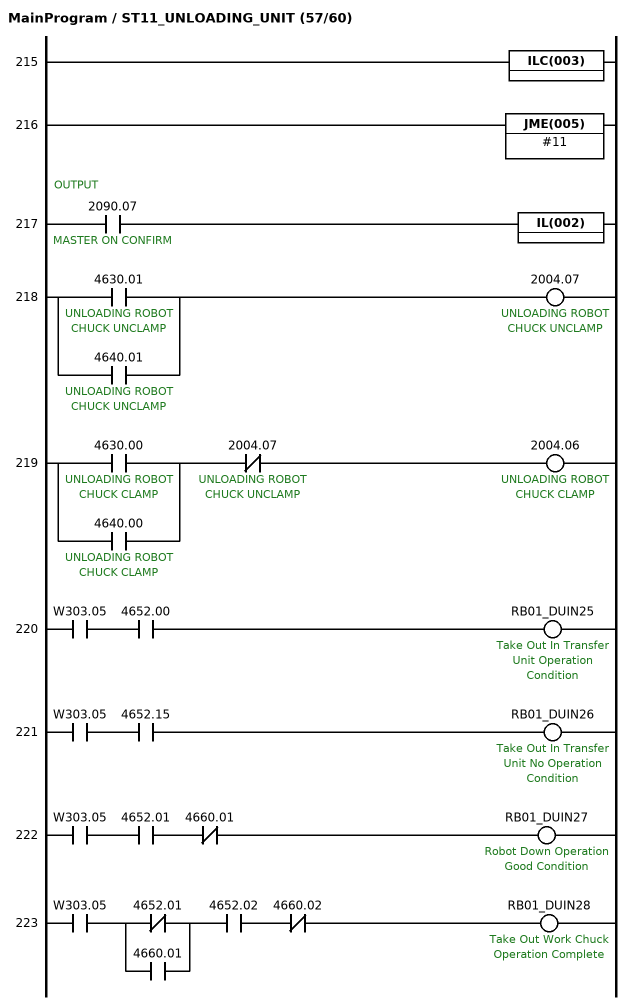
; rung 215
ILC(003)
; rung 216
JME(005) #11
; rung 217: OUTPUT
LD 2090.07  ; MASTER ON CONFIRM
IL(002)
; rung 218
LD 4630.01  ; UNLOADING ROBOT CHUCK UNCLAMP
OR 4640.01  ; UNLOADING ROBOT CHUCK UNCLAMP
OUT 2004.07  ; UNLOADING ROBOT CHUCK UNCLAMP
; rung 219
LD 4630.00  ; UNLOADING ROBOT CHUCK CLAMP
OR 4640.00  ; UNLOADING ROBOT CHUCK CLAMP
ANDNOT 2004.07  ; UNLOADING ROBOT CHUCK UNCLAMP
OUT 2004.06  ; UNLOADING ROBOT CHUCK CLAMP
; rung 220
LD W303.05
AND 4652.00
OUT RB01_DUIN25  ; Take Out In Transfer Unit Operation Condition
; rung 221
LD W303.05
AND 4652.15
OUT RB01_DUIN26  ; Take Out In Transfer Unit No Operation Condition
; rung 222
LD W303.05
AND 4652.01
ANDNOT 4660.01
OUT RB01_DUIN27  ; Robot Down Operation Good Condition
; rung 223
LD W303.05
LDNOT 4652.01
OR 4660.01
ANDLD
AND 4652.02
ANDNOT 4660.02
OUT RB01_DUIN28  ; Take Out Work Chuck  Operation Complete

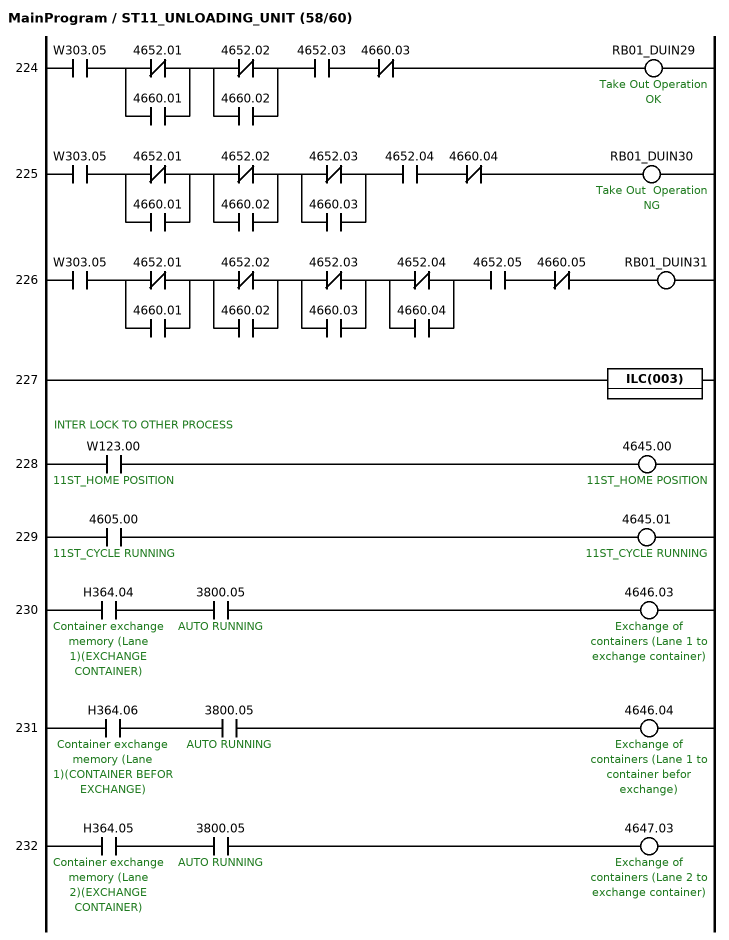
; rung 224
LD W303.05
LDNOT 4652.01
OR 4660.01
ANDLD
LDNOT 4652.02
OR 4660.02
ANDLD
AND 4652.03
ANDNOT 4660.03
OUT RB01_DUIN29  ; Take Out Operation OK
; rung 225
LD W303.05
LDNOT 4652.01
OR 4660.01
ANDLD
LDNOT 4652.02
OR 4660.02
ANDLD
LDNOT 4652.03
OR 4660.03
ANDLD
AND 4652.04
ANDNOT 4660.04
OUT RB01_DUIN30  ; Take Out  Operation NG
; rung 226
LD W303.05
LDNOT 4652.01
OR 4660.01
ANDLD
LDNOT 4652.02
OR 4660.02
ANDLD
LDNOT 4652.03
OR 4660.03
ANDLD
LDNOT 4652.04
OR 4660.04
ANDLD
AND 4652.05
ANDNOT 4660.05
OUT RB01_DUIN31
; rung 227
ILC(003)
; rung 228: INTER LOCK TO OTHER PROCESS
LD W123.00  ; 11ST_HOME POSITION
OUT 4645.00  ; 11ST_HOME POSITION
; rung 229
LD 4605.00  ; 11ST_CYCLE RUNNING
OUT 4645.01  ; 11ST_CYCLE RUNNING
; rung 230
LD H364.04  ; Container exchange memory (Lane 1)(EXCHANGE CONTAINER)
AND 3800.05  ; AUTO RUNNING
OUT 4646.03  ; Exchange of containers (Lane 1 to exchange container)
; rung 231
LD H364.06  ; Container exchange memory (Lane 1)(CONTAINER BEFOR EXCHANGE)
AND 3800.05  ; AUTO RUNNING
OUT 4646.04  ; Exchange of containers (Lane 1 to container befor exchange)
; rung 232
LD H364.05  ; Container exchange memory (Lane 2)(EXCHANGE CONTAINER)
AND 3800.05  ; AUTO RUNNING
OUT 4647.03  ; Exchange of containers (Lane 2 to exchange container)

